# EPICS substitutions: apps/svtCtrlApp/Db/crate_r3.substitutions
# SVT HFCB HV & LV wiener modules substitution file
#  for iseg (HV) MX is slot # 1-10
file iocsoftsvtAppsV/db/iseg.db {
pattern { HOST, MX }
  {"vmetlsvt4","8"}
  {"vmetlsvt4","9"}
  {"vmetlsvt4","10"}
}
#  for mpv (LV) MX is slot # 0-9
file iocsoftsvtAppsV/db/mpv.db {
   pattern { HOST, MX }
  {"vmetlsvt3","0"}
  {"vmetlsvt3","1"}
  {"vmetlsvt3","2"}
  {"vmetlsvt3","3"}
  {"vmetlsvt3","4"}
  {"vmetlsvt3","5"}
  {"vmetlsvt3","6"}
  {"vmetlsvt3","7"}
  {"vmetlsvt3","8"}
}
